(* Logix 5000 project; controller cow Emulate 5570 rev 36.11; software revision 36.00; part 4 of 6 *)
(* tags used below, declared in another part *)
   B126RPM : Speed_RPM;
   B280_Delay : TIMER;
   Cow_SYS_B : System_Data;
   Cow_SYS_D : System_Data;
   SYS_ON : BOOL;
   B111 : MotorX;
   B113 : MotorX;
   B116 : MotorX;
   B126 : MotorX;
   B160 : MotorX;
   B280 : Divider;
   B353 : Gate;
   B354 : Gate;
   B361 : Branch_SV2;
   B362 : Branch_SV2;
   B363 : Branch_SV2;
   B364 : Branch_SV2;
   B365 : Branch_SV2;
   B367 : Branch_SV2;
   B410 : MotorX;
   B420 : MotorX;
   Bin01 : ALIAS FOR rcp_Big_Bin[0];
   Bin02 : ALIAS FOR rcp_Big_Bin[1];
   Bin03 : ALIAS FOR rcp_Big_Bin[2];
   Bin04 : ALIAS FOR rcp_Big_Bin[3];
   Bin05 : ALIAS FOR rcp_Big_Bin[4];
   Bin06 : ALIAS FOR rcp_Big_Bin[5];
   Bin07 : ALIAS FOR rcp_Big_Bin[6];
   Bin08 : ALIAS FOR rcp_Big_Bin[7];
   Bin09 : ALIAS FOR rcp_Big_Bin[8];
   Bin10 : ALIAS FOR rcp_Big_Bin[9];
   Bin11 : ALIAS FOR rcp_Big_Bin[10];
   Bin12 : ALIAS FOR rcp_Big_Bin[11];
   Bin13 : ALIAS FOR rcp_Big_Bin[12];
   Bin14 : ALIAS FOR rcp_Big_Bin[13];
   Bin15 : ALIAS FOR rcp_Big_Bin[14];
   Bin16 : ALIAS FOR rcp_Big_Bin[15];
   D121 : MotorX;
   D162 : MotorX;
   D163 : MotorX;
   D164 : MotorX;
   D230 : MotorX;
   D361 : Branch_SV2;
   D380 : MotorX;
   D411 : MotorX;
   D421 : MotorX;
   STS : INT[100];
   SYS : System_Common;
   SYS_B : Sys_Data;
   SYS_B_DELAY : TIMER;
   SYS_D : Sys_Data;
(* MainProgram, continued *)

ROUTINE B_Intake   (* ladder *)
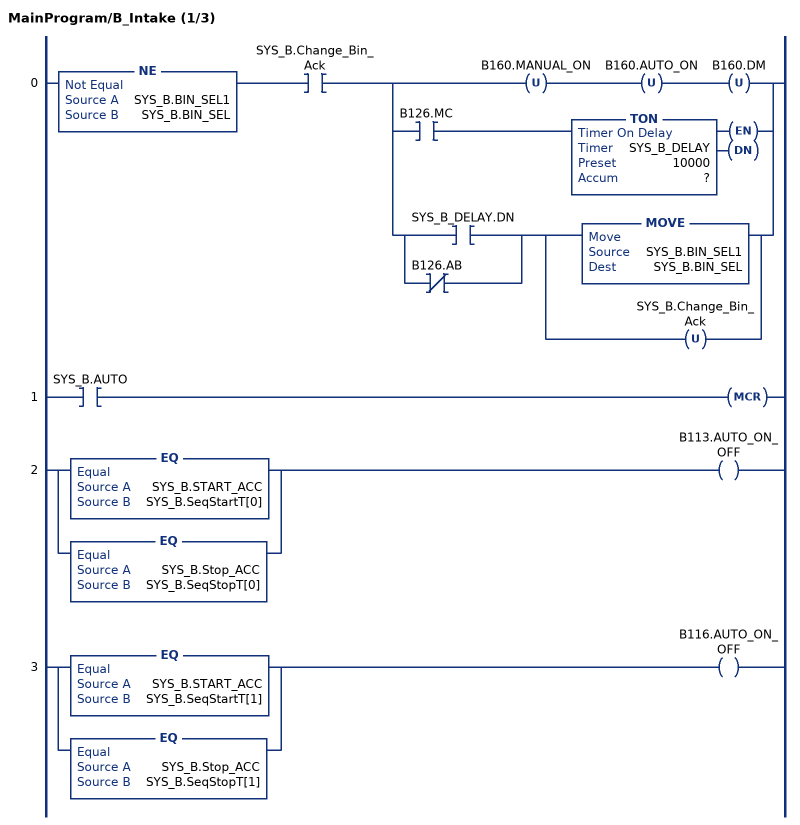
   0: NE(SYS_B.BIN_SEL1,SYS_B.BIN_SEL)XIC(SYS_B.Change_Bin_Ack)[OTU(B160.MANUAL_ON) OTU(B160.AUTO_ON) OTU(B160.DM) ,XIC(B126.MC) TON(SYS_B_DELAY,?,?) ,[XIC(SYS_B_DELAY.DN) ,XIO(B126.AB) ] [MOVE(SYS_B.BIN_SEL1,SYS_B.BIN_SEL) ,OTU(SYS_B.Change_Bin_Ack) ] ];
   1: XIC(SYS_B.AUTO)MCR();
   2: [EQ(SYS_B.START_ACC,SYS_B.SeqStartT[0]) ,EQ(SYS_B.Stop_ACC,SYS_B.SeqStopT[0]) ]OTE(B113.AUTO_ON_OFF);
   3: [EQ(SYS_B.START_ACC,SYS_B.SeqStartT[1]) ,EQ(SYS_B.Stop_ACC,SYS_B.SeqStopT[1]) ]OTE(B116.AUTO_ON_OFF);
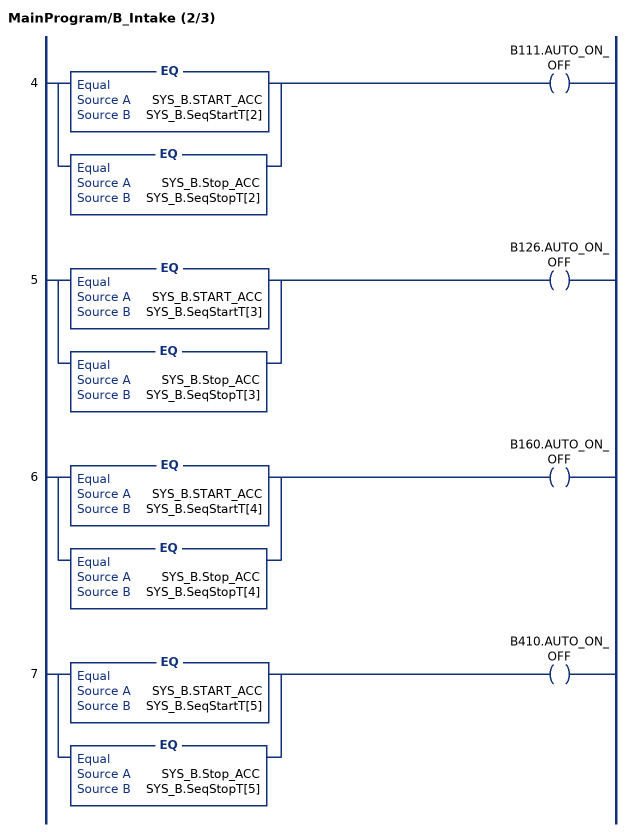
   4: [EQ(SYS_B.START_ACC,SYS_B.SeqStartT[2]) ,EQ(SYS_B.Stop_ACC,SYS_B.SeqStopT[2]) ]OTE(B111.AUTO_ON_OFF);
   5: [EQ(SYS_B.START_ACC,SYS_B.SeqStartT[3]) ,EQ(SYS_B.Stop_ACC,SYS_B.SeqStopT[3]) ]OTE(B126.AUTO_ON_OFF);
   6: [EQ(SYS_B.START_ACC,SYS_B.SeqStartT[4]) ,EQ(SYS_B.Stop_ACC,SYS_B.SeqStopT[4]) ]OTE(B160.AUTO_ON_OFF);
   7: [EQ(SYS_B.START_ACC,SYS_B.SeqStartT[5]) ,EQ(SYS_B.Stop_ACC,SYS_B.SeqStopT[5]) ]OTE(B410.AUTO_ON_OFF);
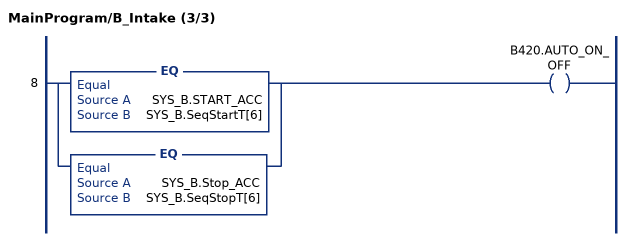
   8: [EQ(SYS_B.START_ACC,SYS_B.SeqStartT[6]) ,EQ(SYS_B.Stop_ACC,SYS_B.SeqStopT[6]) ]OTE(B420.AUTO_ON_OFF);
END_ROUTINE

ROUTINE Device_B   (* ladder *)
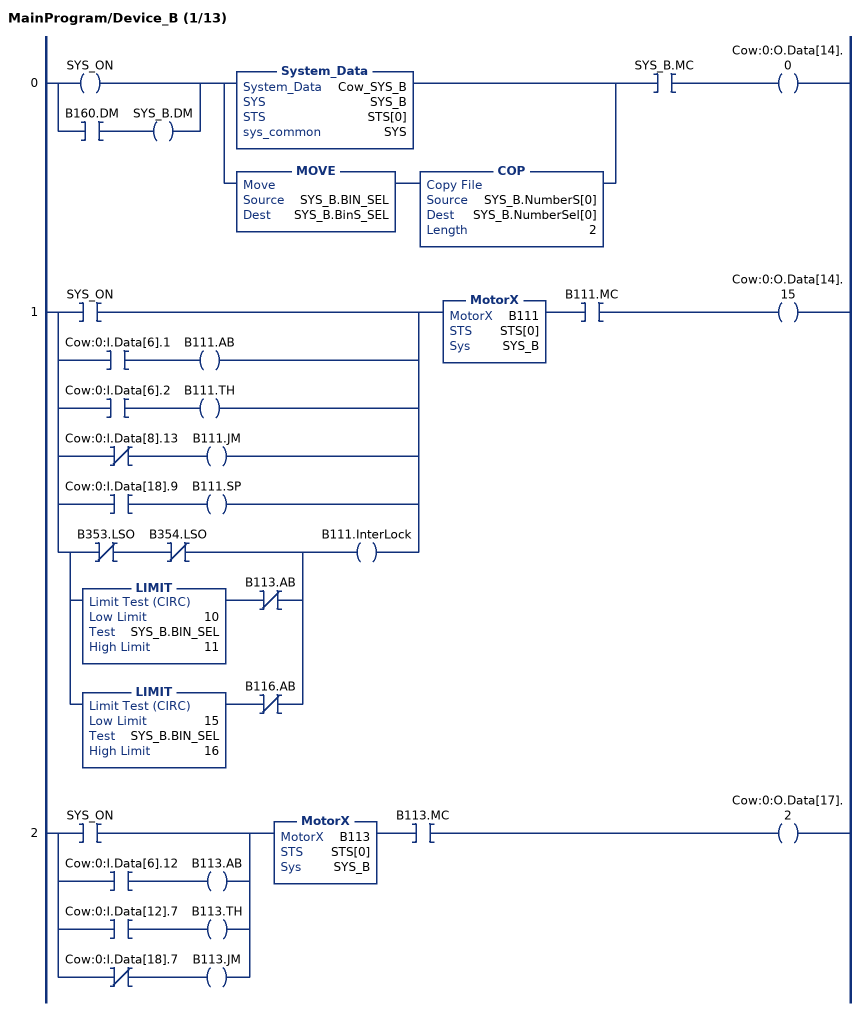
   0: [OTE(SYS_ON) ,XIC(B160.DM) OTE(SYS_B.DM) ][System_Data(Cow_SYS_B,SYS_B,STS[0],SYS) ,MOVE(SYS_B.BIN_SEL,SYS_B.BinS_SEL) COP(SYS_B.NumberS[0],SYS_B.NumberSel[0],2) ]XIC(SYS_B.MC)OTE(Cow:0:O.Data[14].0);
   1: [XIC(SYS_ON) ,XIC(Cow:0:I.Data[6].1) OTE(B111.AB) ,XIC(Cow:0:I.Data[6].2) OTE(B111.TH) ,XIO(Cow:0:I.Data[8].13) OTE(B111.JM) ,XIC(Cow:0:I.Data[18].9) OTE(B111.SP) ,[XIO(B353.LSO) XIO(B354.LSO) ,LIMIT(10,SYS_B.BIN_SEL,11) XIO(B113.AB) ,LIMIT(15,SYS_B.BIN_SEL,16) XIO(B116.AB) ] OTE(B111.InterLock) ]MotorX(B111,STS[0],SYS_B)XIC(B111.MC)OTE(Cow:0:O.Data[14].15);
   2: [XIC(SYS_ON) ,XIC(Cow:0:I.Data[6].12) OTE(B113.AB) ,XIC(Cow:0:I.Data[12].7) OTE(B113.TH) ,XIO(Cow:0:I.Data[18].7) OTE(B113.JM) ]MotorX(B113,STS[0],SYS_B)XIC(B113.MC)OTE(Cow:0:O.Data[17].2);
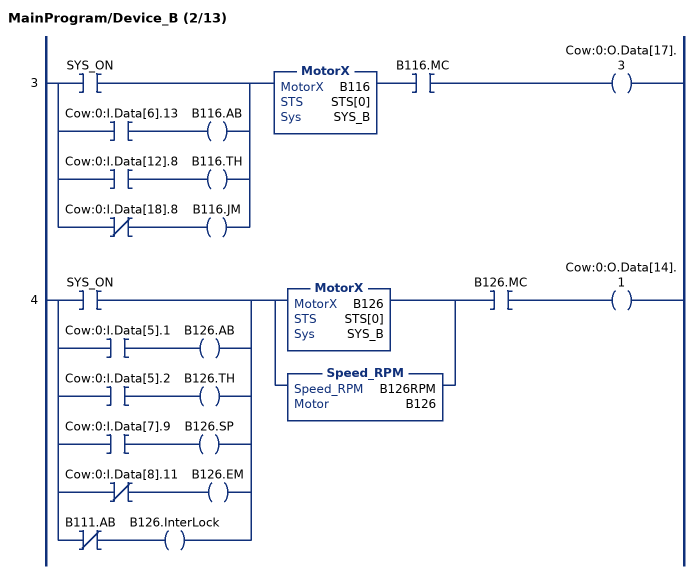
   3: [XIC(SYS_ON) ,XIC(Cow:0:I.Data[6].13) OTE(B116.AB) ,XIC(Cow:0:I.Data[12].8) OTE(B116.TH) ,XIO(Cow:0:I.Data[18].8) OTE(B116.JM) ]MotorX(B116,STS[0],SYS_B)XIC(B116.MC)OTE(Cow:0:O.Data[17].3);
   4: [XIC(SYS_ON) ,XIC(Cow:0:I.Data[5].1) OTE(B126.AB) ,XIC(Cow:0:I.Data[5].2) OTE(B126.TH) ,XIC(Cow:0:I.Data[7].9) OTE(B126.SP) ,XIO(Cow:0:I.Data[8].11) OTE(B126.EM) ,XIO(B111.AB) OTE(B126.InterLock) ][MotorX(B126,STS[0],SYS_B) ,Speed_RPM(B126RPM,B126) ]XIC(B126.MC)OTE(Cow:0:O.Data[14].1);
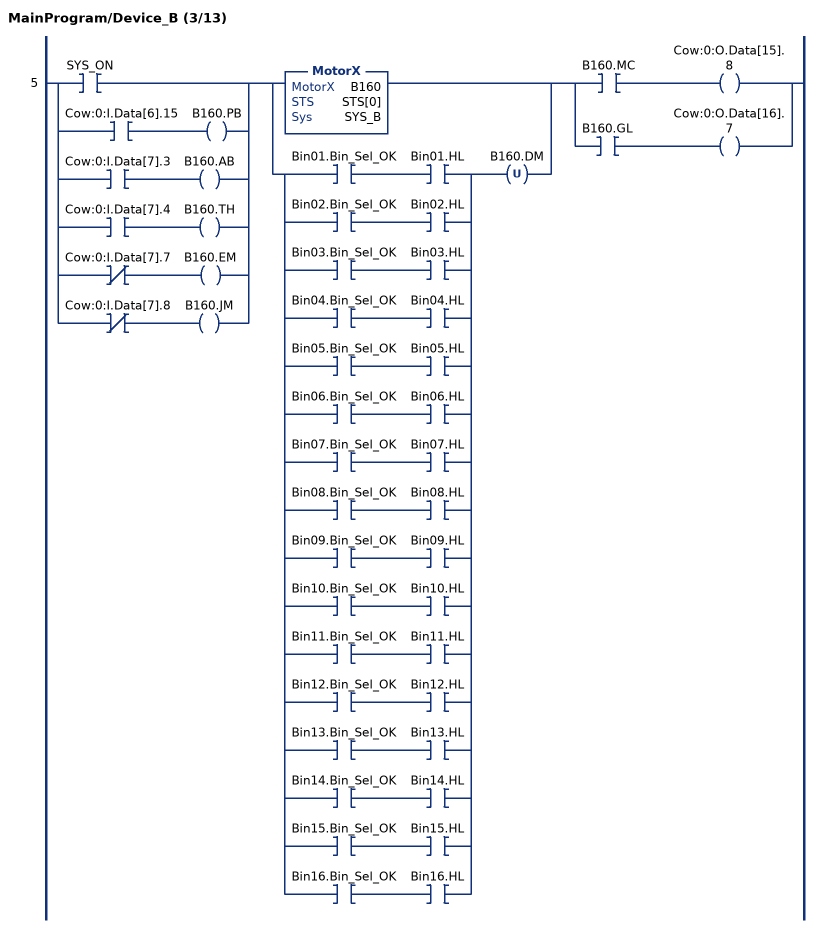
   5: [XIC(SYS_ON) ,XIC(Cow:0:I.Data[6].15) OTE(B160.PB) ,XIC(Cow:0:I.Data[7].3) OTE(B160.AB) ,XIC(Cow:0:I.Data[7].4) OTE(B160.TH) ,XIO(Cow:0:I.Data[7].7) OTE(B160.EM) ,XIO(Cow:0:I.Data[7].8) OTE(B160.JM) ][MotorX(B160,STS[0],SYS_B) ,[XIC(Bin01.Bin_Sel_OK) XIC(Bin01.HL) ,XIC(Bin02.Bin_Sel_OK) XIC(Bin02.HL) ,XIC(Bin03.Bin_Sel_OK) XIC(Bin03.HL) ,XIC(Bin04.Bin_Sel_OK) XIC(Bin04.HL) ,XIC(Bin05.Bin_Sel_OK) XIC(Bin05.HL) ,XIC(Bin06.Bin_Sel_OK) XIC(Bin06.HL) ,XIC(Bin07.Bin_Sel_OK) XIC(Bin07.HL) ,XIC(Bin08.Bin_Sel_OK) XIC(Bin08.HL) ,XIC(Bin09.Bin_Sel_OK) XIC(Bin09.HL) ,XIC(Bin10.Bin_Sel_OK) XIC(Bin10.HL) ,XIC(Bin11.Bin_Sel_OK) XIC(Bin11.HL) ,XIC(Bin12.Bin_Sel_OK) XIC(Bin12.HL) ,XIC(Bin13.Bin_Sel_OK) XIC(Bin13.HL) ,XIC(Bin14.Bin_Sel_OK) XIC(Bin14.HL) ,XIC(Bin15.Bin_Sel_OK) XIC(Bin15.HL) ,XIC(Bin16.Bin_Sel_OK) XIC(Bin16.HL) ] OTU(B160.DM) ][XIC(B160.MC) OTE(Cow:0:O.Data[15].8) ,XIC(B160.GL) OTE(Cow:0:O.Data[16].7) ];
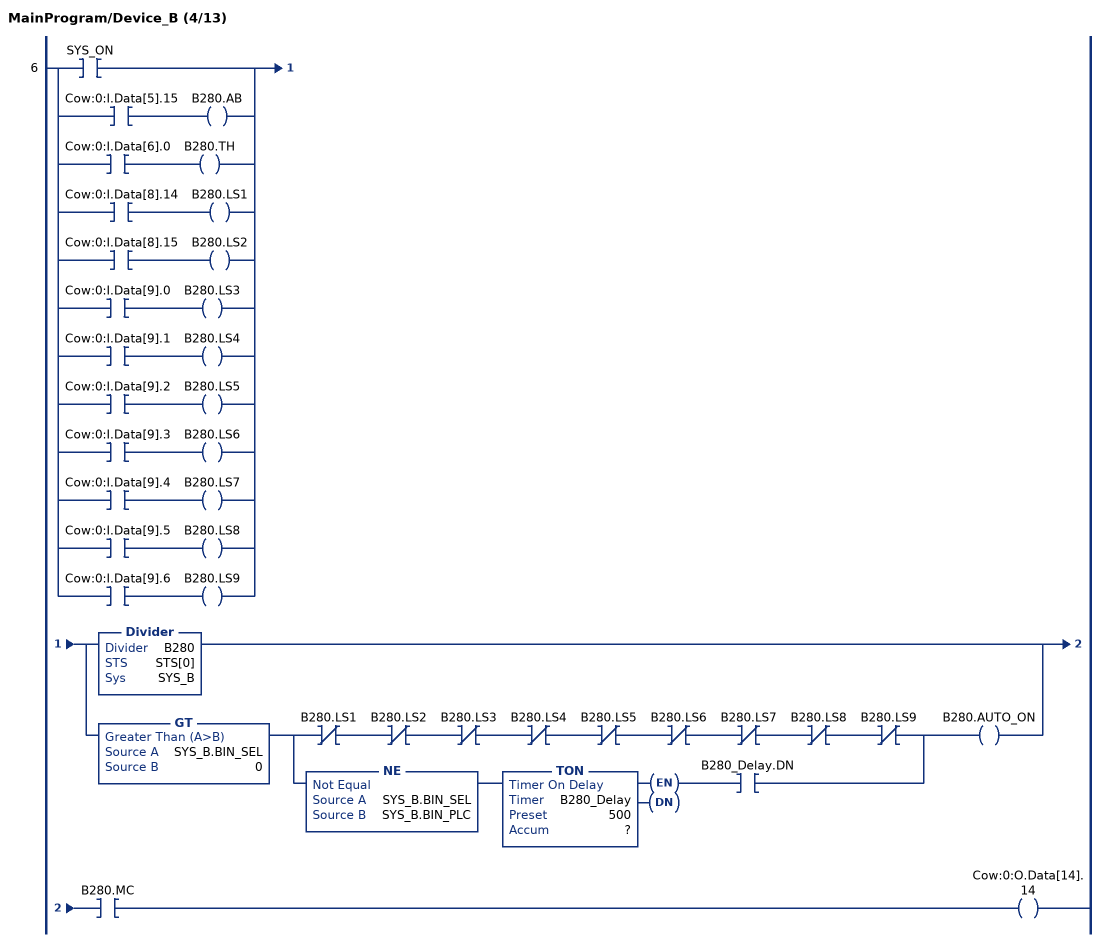
   6: [XIC(SYS_ON) ,XIC(Cow:0:I.Data[5].15) OTE(B280.AB) ,XIC(Cow:0:I.Data[6].0) OTE(B280.TH) ,XIC(Cow:0:I.Data[8].14) OTE(B280.LS1) ,XIC(Cow:0:I.Data[8].15) OTE(B280.LS2) ,XIC(Cow:0:I.Data[9].0) OTE(B280.LS3) ,XIC(Cow:0:I.Data[9].1) OTE(B280.LS4) ,XIC(Cow:0:I.Data[9].2) OTE(B280.LS5) ,XIC(Cow:0:I.Data[9].3) OTE(B280.LS6) ,XIC(Cow:0:I.Data[9].4) OTE(B280.LS7) ,XIC(Cow:0:I.Data[9].5) OTE(B280.LS8) ,XIC(Cow:0:I.Data[9].6) OTE(B280.LS9) ][Divider(B280,STS[0],SYS_B) ,GT(SYS_B.BIN_SEL,0) [XIO(B280.LS1) XIO(B280.LS2) XIO(B280.LS3) XIO(B280.LS4) XIO(B280.LS5) XIO(B280.LS6) XIO(B280.LS7) XIO(B280.LS8) XIO(B280.LS9) ,NE(SYS_B.BIN_SEL,SYS_B.BIN_PLC) TON(B280_Delay,?,?) XIC(B280_Delay.DN) ] OTE(B280.AUTO_ON) ]XIC(B280.MC)OTE(Cow:0:O.Data[14].14);
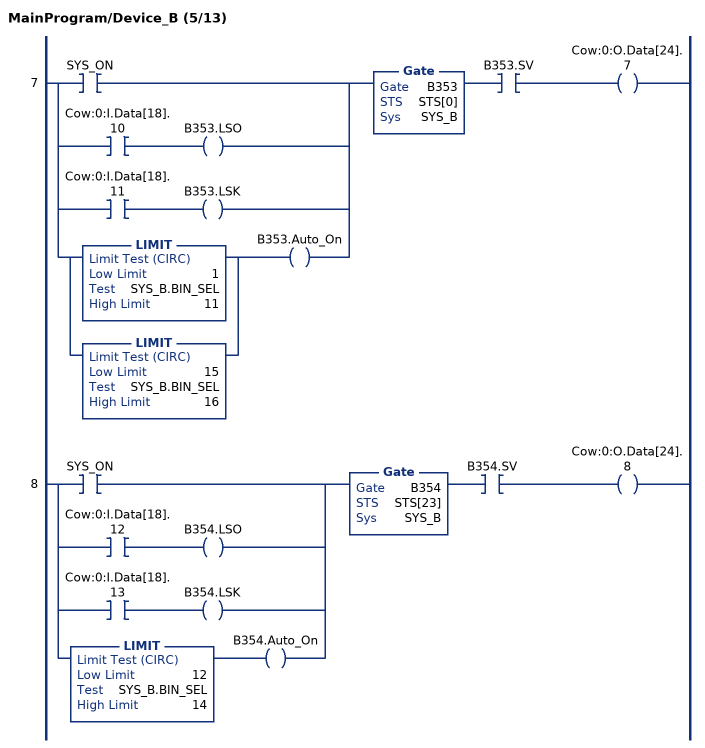
   7: [XIC(SYS_ON) ,XIC(Cow:0:I.Data[18].10) OTE(B353.LSO) ,XIC(Cow:0:I.Data[18].11) OTE(B353.LSK) ,[LIMIT(1,SYS_B.BIN_SEL,11) ,LIMIT(15,SYS_B.BIN_SEL,16) ] OTE(B353.Auto_On) ]Gate(B353,STS[0],SYS_B)XIC(B353.SV)OTE(Cow:0:O.Data[24].7);
   8: [XIC(SYS_ON) ,XIC(Cow:0:I.Data[18].12) OTE(B354.LSO) ,XIC(Cow:0:I.Data[18].13) OTE(B354.LSK) ,LIMIT(12,SYS_B.BIN_SEL,14) OTE(B354.Auto_On) ]Gate(B354,STS[23],SYS_B)XIC(B354.SV)OTE(Cow:0:O.Data[24].8);
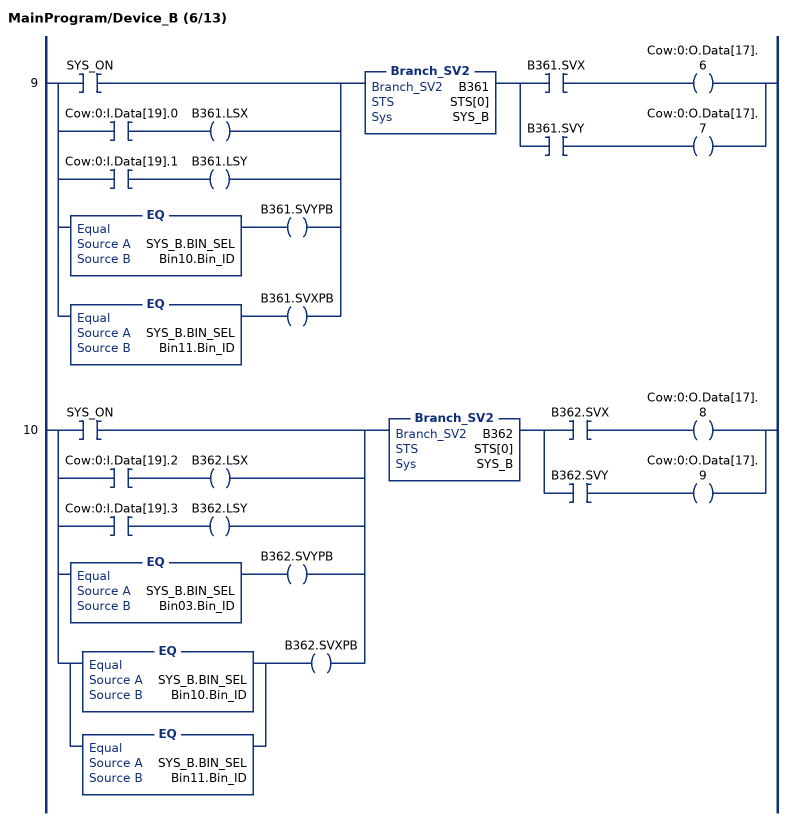
   9: [XIC(SYS_ON) ,XIC(Cow:0:I.Data[19].0) OTE(B361.LSX) ,XIC(Cow:0:I.Data[19].1) OTE(B361.LSY) ,EQ(SYS_B.BIN_SEL,Bin10.Bin_ID) OTE(B361.SVYPB) ,EQ(SYS_B.BIN_SEL,Bin11.Bin_ID) OTE(B361.SVXPB) ]Branch_SV2(B361,STS[0],SYS_B)[XIC(B361.SVX) OTE(Cow:0:O.Data[17].6) ,XIC(B361.SVY) OTE(Cow:0:O.Data[17].7) ];
   10: [XIC(SYS_ON) ,XIC(Cow:0:I.Data[19].2) OTE(B362.LSX) ,XIC(Cow:0:I.Data[19].3) OTE(B362.LSY) ,EQ(SYS_B.BIN_SEL,Bin03.Bin_ID) OTE(B362.SVYPB) ,[EQ(SYS_B.BIN_SEL,Bin10.Bin_ID) ,EQ(SYS_B.BIN_SEL,Bin11.Bin_ID) ] OTE(B362.SVXPB) ]Branch_SV2(B362,STS[0],SYS_B)[XIC(B362.SVX) OTE(Cow:0:O.Data[17].8) ,XIC(B362.SVY) OTE(Cow:0:O.Data[17].9) ];
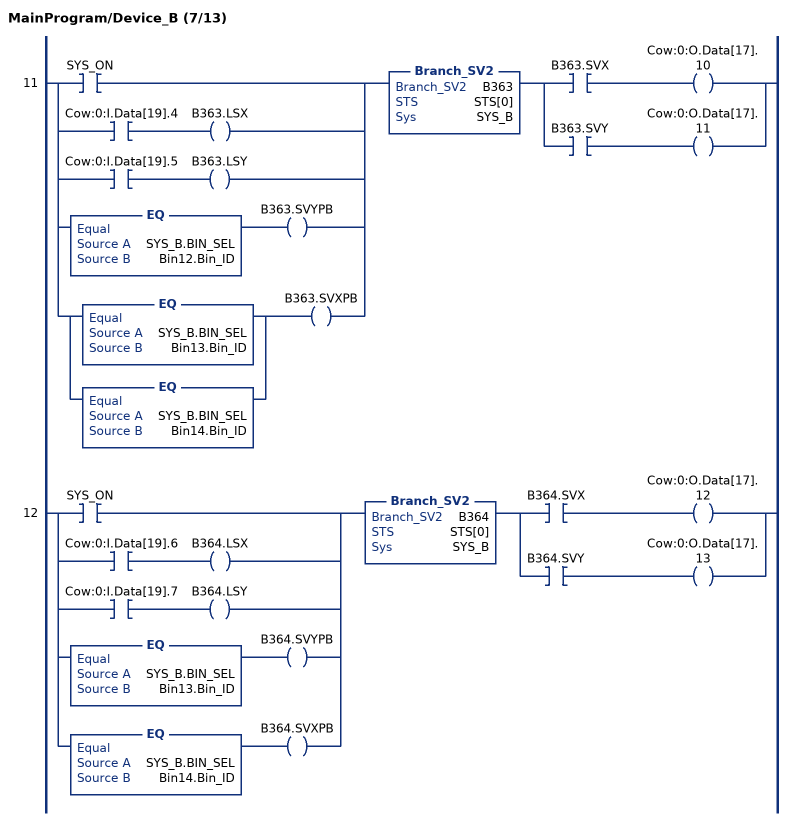
   11: [XIC(SYS_ON) ,XIC(Cow:0:I.Data[19].4) OTE(B363.LSX) ,XIC(Cow:0:I.Data[19].5) OTE(B363.LSY) ,EQ(SYS_B.BIN_SEL,Bin12.Bin_ID) OTE(B363.SVYPB) ,[EQ(SYS_B.BIN_SEL,Bin13.Bin_ID) ,EQ(SYS_B.BIN_SEL,Bin14.Bin_ID) ] OTE(B363.SVXPB) ]Branch_SV2(B363,STS[0],SYS_B)[XIC(B363.SVX) OTE(Cow:0:O.Data[17].10) ,XIC(B363.SVY) OTE(Cow:0:O.Data[17].11) ];
   12: [XIC(SYS_ON) ,XIC(Cow:0:I.Data[19].6) OTE(B364.LSX) ,XIC(Cow:0:I.Data[19].7) OTE(B364.LSY) ,EQ(SYS_B.BIN_SEL,Bin13.Bin_ID) OTE(B364.SVYPB) ,EQ(SYS_B.BIN_SEL,Bin14.Bin_ID) OTE(B364.SVXPB) ]Branch_SV2(B364,STS[0],SYS_B)[XIC(B364.SVX) OTE(Cow:0:O.Data[17].12) ,XIC(B364.SVY) OTE(Cow:0:O.Data[17].13) ];
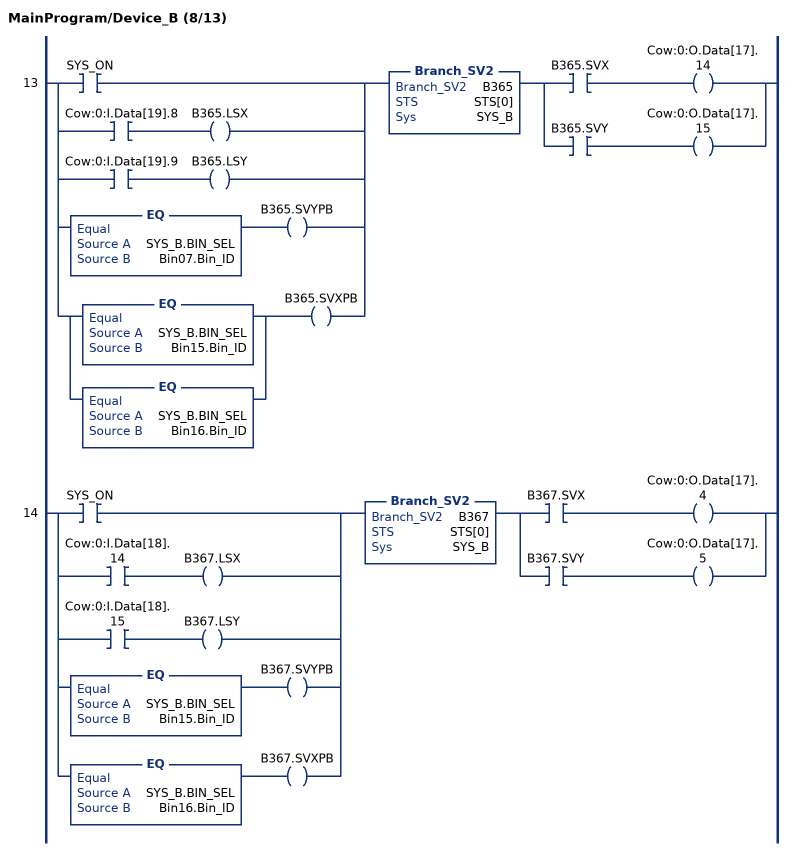
   13: [XIC(SYS_ON) ,XIC(Cow:0:I.Data[19].8) OTE(B365.LSX) ,XIC(Cow:0:I.Data[19].9) OTE(B365.LSY) ,EQ(SYS_B.BIN_SEL,Bin07.Bin_ID) OTE(B365.SVYPB) ,[EQ(SYS_B.BIN_SEL,Bin15.Bin_ID) ,EQ(SYS_B.BIN_SEL,Bin16.Bin_ID) ] OTE(B365.SVXPB) ]Branch_SV2(B365,STS[0],SYS_B)[XIC(B365.SVX) OTE(Cow:0:O.Data[17].14) ,XIC(B365.SVY) OTE(Cow:0:O.Data[17].15) ];
   14: [XIC(SYS_ON) ,XIC(Cow:0:I.Data[18].14) OTE(B367.LSX) ,XIC(Cow:0:I.Data[18].15) OTE(B367.LSY) ,EQ(SYS_B.BIN_SEL,Bin15.Bin_ID) OTE(B367.SVYPB) ,EQ(SYS_B.BIN_SEL,Bin16.Bin_ID) OTE(B367.SVXPB) ]Branch_SV2(B367,STS[0],SYS_B)[XIC(B367.SVX) OTE(Cow:0:O.Data[17].4) ,XIC(B367.SVY) OTE(Cow:0:O.Data[17].5) ];
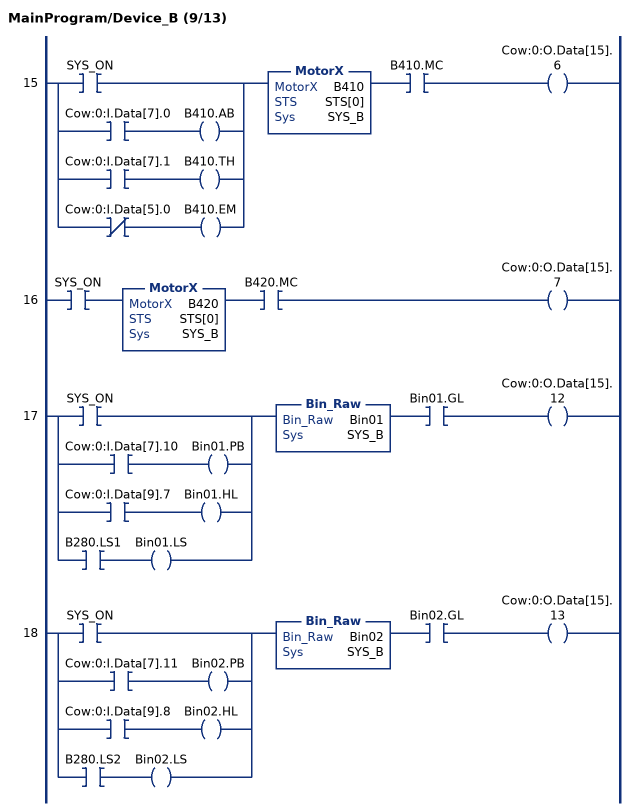
   15: [XIC(SYS_ON) ,XIC(Cow:0:I.Data[7].0) OTE(B410.AB) ,XIC(Cow:0:I.Data[7].1) OTE(B410.TH) ,XIO(Cow:0:I.Data[5].0) OTE(B410.EM) ]MotorX(B410,STS[0],SYS_B)XIC(B410.MC)OTE(Cow:0:O.Data[15].6);
   16: XIC(SYS_ON)MotorX(B420,STS[0],SYS_B)XIC(B420.MC)OTE(Cow:0:O.Data[15].7);
   17: [XIC(SYS_ON) ,XIC(Cow:0:I.Data[7].10) OTE(Bin01.PB) ,XIC(Cow:0:I.Data[9].7) OTE(Bin01.HL) ,XIC(B280.LS1) OTE(Bin01.LS) ]Bin_Raw(Bin01,SYS_B)XIC(Bin01.GL)OTE(Cow:0:O.Data[15].12);
   18: [XIC(SYS_ON) ,XIC(Cow:0:I.Data[7].11) OTE(Bin02.PB) ,XIC(Cow:0:I.Data[9].8) OTE(Bin02.HL) ,XIC(B280.LS2) OTE(Bin02.LS) ]Bin_Raw(Bin02,SYS_B)XIC(Bin02.GL)OTE(Cow:0:O.Data[15].13);
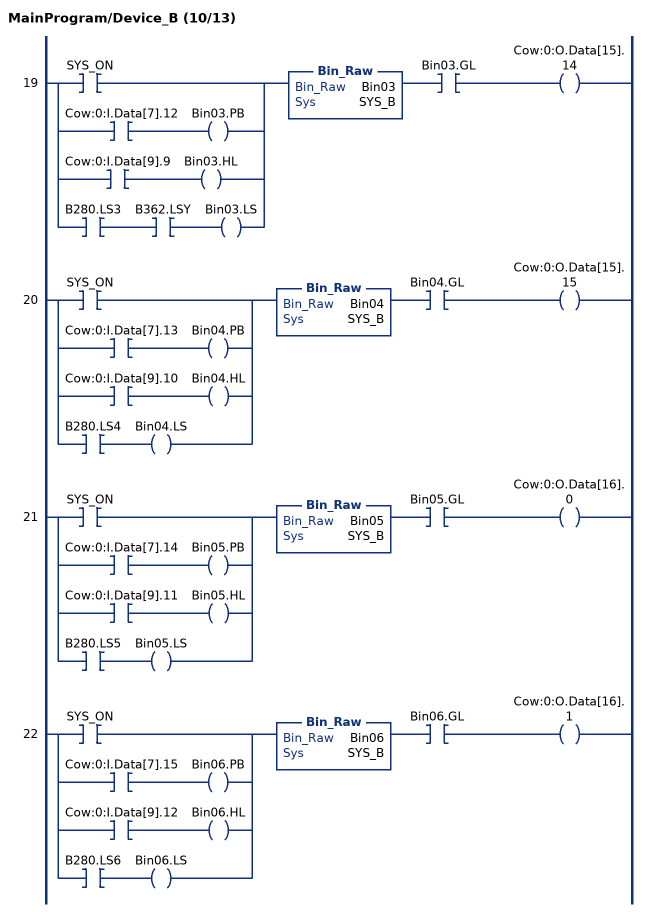
   19: [XIC(SYS_ON) ,XIC(Cow:0:I.Data[7].12) OTE(Bin03.PB) ,XIC(Cow:0:I.Data[9].9) OTE(Bin03.HL) ,XIC(B280.LS3) XIC(B362.LSY) OTE(Bin03.LS) ]Bin_Raw(Bin03,SYS_B)XIC(Bin03.GL)OTE(Cow:0:O.Data[15].14);
   20: [XIC(SYS_ON) ,XIC(Cow:0:I.Data[7].13) OTE(Bin04.PB) ,XIC(Cow:0:I.Data[9].10) OTE(Bin04.HL) ,XIC(B280.LS4) OTE(Bin04.LS) ]Bin_Raw(Bin04,SYS_B)XIC(Bin04.GL)OTE(Cow:0:O.Data[15].15);
   21: [XIC(SYS_ON) ,XIC(Cow:0:I.Data[7].14) OTE(Bin05.PB) ,XIC(Cow:0:I.Data[9].11) OTE(Bin05.HL) ,XIC(B280.LS5) OTE(Bin05.LS) ]Bin_Raw(Bin05,SYS_B)XIC(Bin05.GL)OTE(Cow:0:O.Data[16].0);
   22: [XIC(SYS_ON) ,XIC(Cow:0:I.Data[7].15) OTE(Bin06.PB) ,XIC(Cow:0:I.Data[9].12) OTE(Bin06.HL) ,XIC(B280.LS6) OTE(Bin06.LS) ]Bin_Raw(Bin06,SYS_B)XIC(Bin06.GL)OTE(Cow:0:O.Data[16].1);
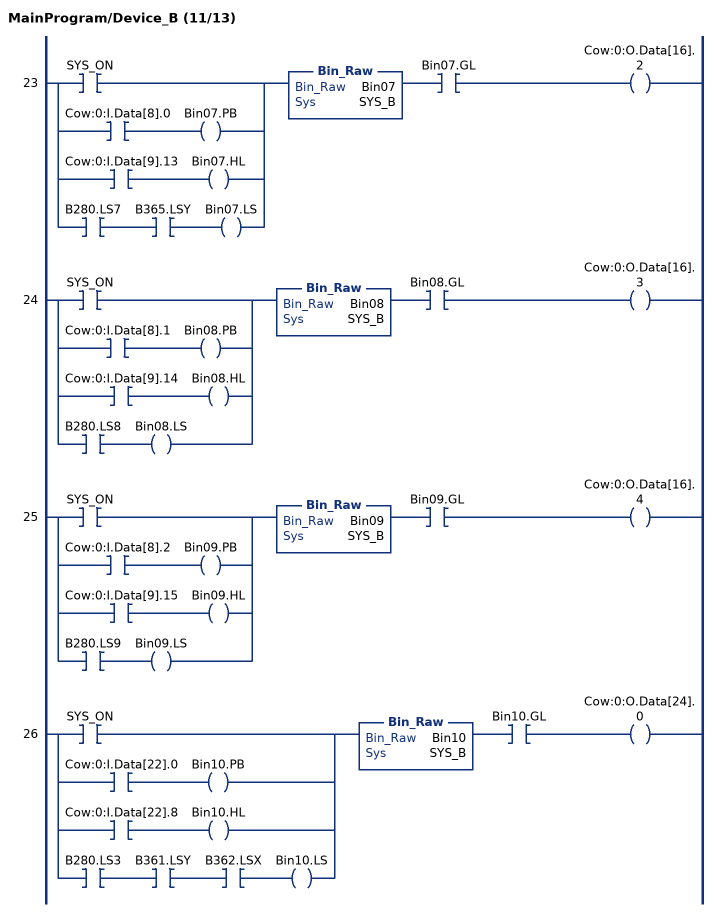
   23: [XIC(SYS_ON) ,XIC(Cow:0:I.Data[8].0) OTE(Bin07.PB) ,XIC(Cow:0:I.Data[9].13) OTE(Bin07.HL) ,XIC(B280.LS7) XIC(B365.LSY) OTE(Bin07.LS) ]Bin_Raw(Bin07,SYS_B)XIC(Bin07.GL)OTE(Cow:0:O.Data[16].2);
   24: [XIC(SYS_ON) ,XIC(Cow:0:I.Data[8].1) OTE(Bin08.PB) ,XIC(Cow:0:I.Data[9].14) OTE(Bin08.HL) ,XIC(B280.LS8) OTE(Bin08.LS) ]Bin_Raw(Bin08,SYS_B)XIC(Bin08.GL)OTE(Cow:0:O.Data[16].3);
   25: [XIC(SYS_ON) ,XIC(Cow:0:I.Data[8].2) OTE(Bin09.PB) ,XIC(Cow:0:I.Data[9].15) OTE(Bin09.HL) ,XIC(B280.LS9) OTE(Bin09.LS) ]Bin_Raw(Bin09,SYS_B)XIC(Bin09.GL)OTE(Cow:0:O.Data[16].4);
   26: [XIC(SYS_ON) ,XIC(Cow:0:I.Data[22].0) OTE(Bin10.PB) ,XIC(Cow:0:I.Data[22].8) OTE(Bin10.HL) ,XIC(B280.LS3) XIC(B361.LSY) XIC(B362.LSX) OTE(Bin10.LS) ]Bin_Raw(Bin10,SYS_B)XIC(Bin10.GL)OTE(Cow:0:O.Data[24].0);
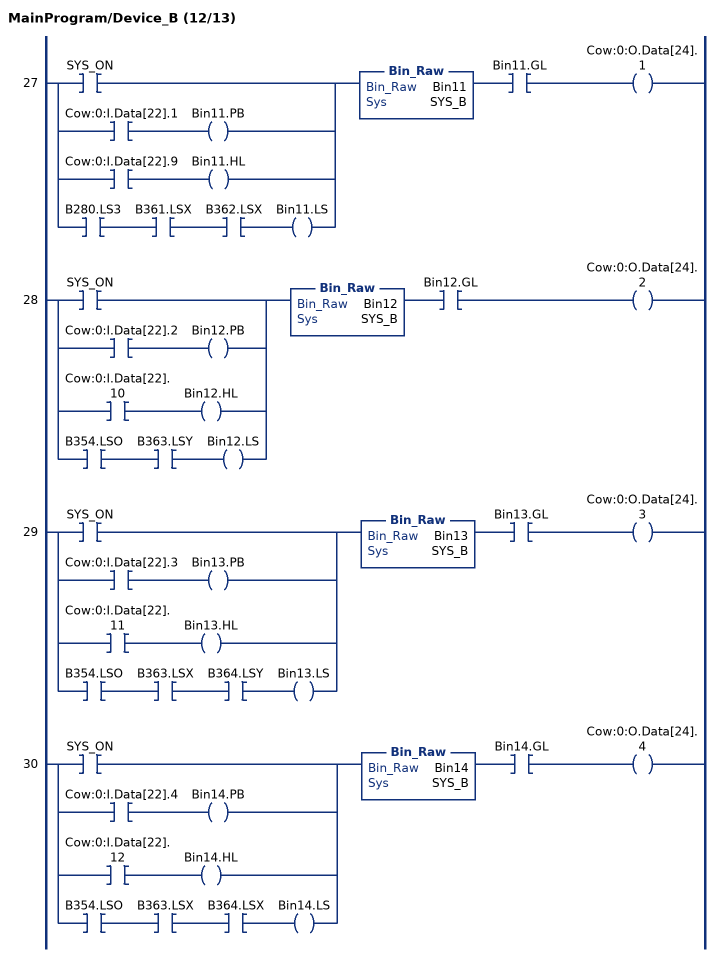
   27: [XIC(SYS_ON) ,XIC(Cow:0:I.Data[22].1) OTE(Bin11.PB) ,XIC(Cow:0:I.Data[22].9) OTE(Bin11.HL) ,XIC(B280.LS3) XIC(B361.LSX) XIC(B362.LSX) OTE(Bin11.LS) ]Bin_Raw(Bin11,SYS_B)XIC(Bin11.GL)OTE(Cow:0:O.Data[24].1);
   28: [XIC(SYS_ON) ,XIC(Cow:0:I.Data[22].2) OTE(Bin12.PB) ,XIC(Cow:0:I.Data[22].10) OTE(Bin12.HL) ,XIC(B354.LSO) XIC(B363.LSY) OTE(Bin12.LS) ]Bin_Raw(Bin12,SYS_B)XIC(Bin12.GL)OTE(Cow:0:O.Data[24].2);
   29: [XIC(SYS_ON) ,XIC(Cow:0:I.Data[22].3) OTE(Bin13.PB) ,XIC(Cow:0:I.Data[22].11) OTE(Bin13.HL) ,XIC(B354.LSO) XIC(B363.LSX) XIC(B364.LSY) OTE(Bin13.LS) ]Bin_Raw(Bin13,SYS_B)XIC(Bin13.GL)OTE(Cow:0:O.Data[24].3);
   30: [XIC(SYS_ON) ,XIC(Cow:0:I.Data[22].4) OTE(Bin14.PB) ,XIC(Cow:0:I.Data[22].12) OTE(Bin14.HL) ,XIC(B354.LSO) XIC(B363.LSX) XIC(B364.LSX) OTE(Bin14.LS) ]Bin_Raw(Bin14,SYS_B)XIC(Bin14.GL)OTE(Cow:0:O.Data[24].4);
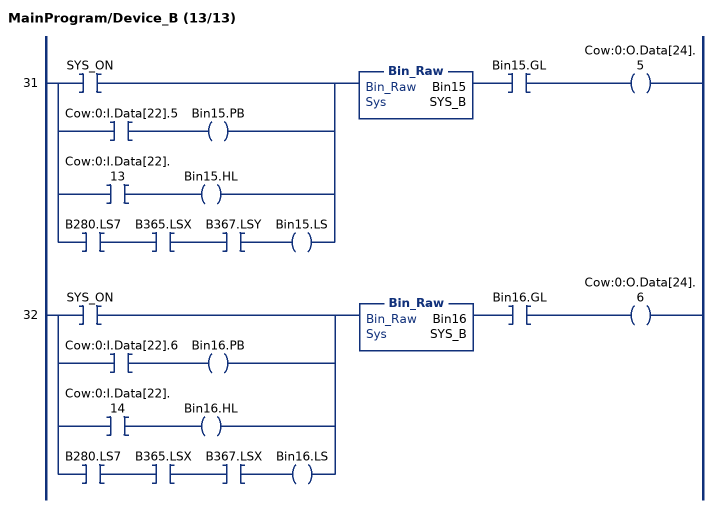
   31: [XIC(SYS_ON) ,XIC(Cow:0:I.Data[22].5) OTE(Bin15.PB) ,XIC(Cow:0:I.Data[22].13) OTE(Bin15.HL) ,XIC(B280.LS7) XIC(B365.LSX) XIC(B367.LSY) OTE(Bin15.LS) ]Bin_Raw(Bin15,SYS_B)XIC(Bin15.GL)OTE(Cow:0:O.Data[24].5);
   32: [XIC(SYS_ON) ,XIC(Cow:0:I.Data[22].6) OTE(Bin16.PB) ,XIC(Cow:0:I.Data[22].14) OTE(Bin16.HL) ,XIC(B280.LS7) XIC(B365.LSX) XIC(B367.LSX) OTE(Bin16.LS) ]Bin_Raw(Bin16,SYS_B)XIC(Bin16.GL)OTE(Cow:0:O.Data[24].6);
END_ROUTINE

ROUTINE Device_D   (* ladder *)
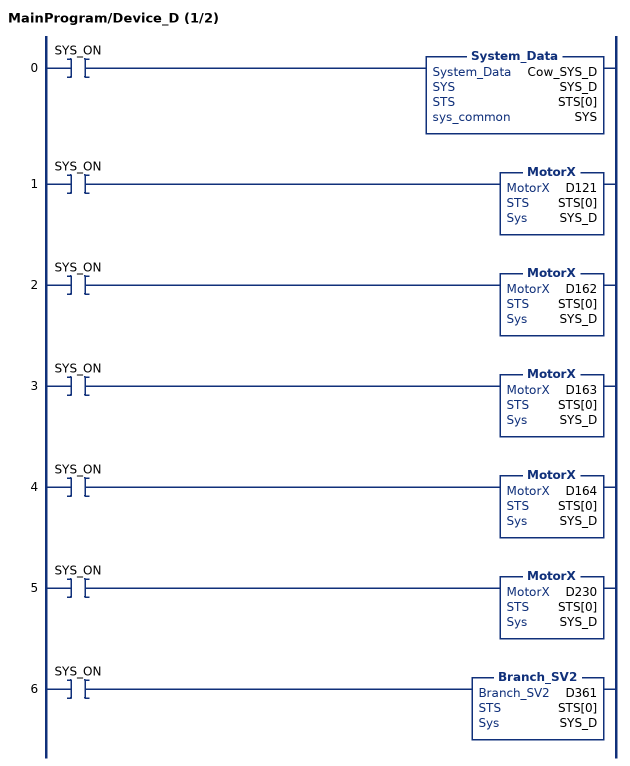
   0: XIC(SYS_ON)System_Data(Cow_SYS_D,SYS_D,STS[0],SYS);
   1: XIC(SYS_ON)MotorX(D121,STS[0],SYS_D);
   2: XIC(SYS_ON)MotorX(D162,STS[0],SYS_D);
   3: XIC(SYS_ON)MotorX(D163,STS[0],SYS_D);
   4: XIC(SYS_ON)MotorX(D164,STS[0],SYS_D);
   5: XIC(SYS_ON)MotorX(D230,STS[0],SYS_D);
   6: XIC(SYS_ON)Branch_SV2(D361,STS[0],SYS_D);
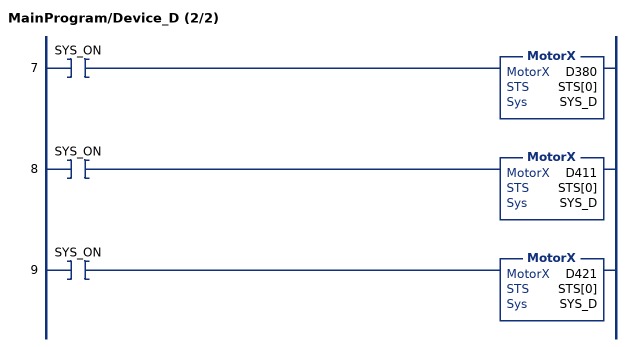
   7: XIC(SYS_ON)MotorX(D380,STS[0],SYS_D);
   8: XIC(SYS_ON)MotorX(D411,STS[0],SYS_D);
   9: XIC(SYS_ON)MotorX(D421,STS[0],SYS_D);
END_ROUTINE
